PROGRAM PRG_TerminBoxInfo
VAR
END_VAR

//Terminal 0
GVL_IO.dwTerminalInfo[1].fbTerminalInfo(nTerminalState:= 8,
                                        sTerminalState => GVL_IO.dwTerminalInfo[0].sTerminalInfo);
//Terminal 1
GVL_IO.dwTerminalInfo[1].fbTerminalInfo(nTerminalState:= GVL_IO.dwTerminalInfo[1].nTerminal_State,
                                        sTerminalState => GVL_IO.dwTerminalInfo[1].sTerminalInfo);  
//Terminal 2
GVL_IO.dwTerminalInfo[2].fbTerminalInfo(nTerminalState:= GVL_IO.dwTerminalInfo[2].nTerminal_State,
                                        sTerminalState => GVL_IO.dwTerminalInfo[2].sTerminalInfo); 
//Terminal 3
GVL_IO.dwTerminalInfo[3].fbTerminalInfo(nTerminalState:= GVL_IO.dwTerminalInfo[3].nTerminal_State,
                                        sTerminalState => GVL_IO.dwTerminalInfo[3].sTerminalInfo); 
//Terminal 4
GVL_IO.dwTerminalInfo[4].fbTerminalInfo(nTerminalState:= GVL_IO.dwTerminalInfo[4].nTerminal_State,
                                        sTerminalState => GVL_IO.dwTerminalInfo[4].sTerminalInfo); 
//Terminal 5
GVL_IO.dwTerminalInfo[5].fbTerminalInfo(nTerminalState:= GVL_IO.dwTerminalInfo[5].nTerminal_State,
                                        sTerminalState => GVL_IO.dwTerminalInfo[5].sTerminalInfo); 
//Terminal 6
GVL_IO.dwTerminalInfo[6].fbTerminalInfo(nTerminalState:= GVL_IO.dwTerminalInfo[6].nTerminal_State,
                                        sTerminalState => GVL_IO.dwTerminalInfo[6].sTerminalInfo); 
//Terminal 7
GVL_IO.dwTerminalInfo[7].fbTerminalInfo(nTerminalState:= GVL_IO.dwTerminalInfo[7].nTerminal_State,
                                        sTerminalState => GVL_IO.dwTerminalInfo[7].sTerminalInfo); 
//Terminal 8
GVL_IO.dwTerminalInfo[8].fbTerminalInfo(nTerminalState:= GVL_IO.dwTerminalInfo[8].nTerminal_State,
                                        sTerminalState => GVL_IO.dwTerminalInfo[8].sTerminalInfo); 
//Terminal 9
GVL_IO.dwTerminalInfo[9].fbTerminalInfo(nTerminalState:= GVL_IO.dwTerminalInfo[9].nTerminal_State,
                                        sTerminalState => GVL_IO.dwTerminalInfo[9].sTerminalInfo); 
//Terminal 10
GVL_IO.dwTerminalInfo[10].fbTerminalInfo(nTerminalState:= GVL_IO.dwTerminalInfo[10].nTerminal_State,
                                        sTerminalState => GVL_IO.dwTerminalInfo[10].sTerminalInfo); 
//Terminal 11
GVL_IO.dwTerminalInfo[11].fbTerminalInfo(nTerminalState:= GVL_IO.dwTerminalInfo[11].nTerminal_State,
                                        sTerminalState => GVL_IO.dwTerminalInfo[11].sTerminalInfo); 
//Terminal 12
GVL_IO.dwTerminalInfo[12].fbTerminalInfo(nTerminalState:= GVL_IO.dwTerminalInfo[12].nTerminal_State,
                                        sTerminalState => GVL_IO.dwTerminalInfo[12].sTerminalInfo); 										
//Terminal 13
GVL_IO.dwTerminalInfo[13].fbTerminalInfo(nTerminalState:= GVL_IO.dwTerminalInfo[13].nTerminal_State,
                                        sTerminalState => GVL_IO.dwTerminalInfo[13].sTerminalInfo); 
//Terminal 14
GVL_IO.dwTerminalInfo[14].fbTerminalInfo(nTerminalState:= GVL_IO.dwTerminalInfo[14].nTerminal_State,
                                        sTerminalState => GVL_IO.dwTerminalInfo[14].sTerminalInfo);
										
//Terminal 15
GVL_IO.dwTerminalInfo[15].fbTerminalInfo(nTerminalState:= GVL_IO.dwTerminalInfo[15].nTerminal_State,
                                        sTerminalState => GVL_IO.dwTerminalInfo[15].sTerminalInfo); 
//Terminal 16
GVL_IO.dwTerminalInfo[16].fbTerminalInfo(nTerminalState:= 8,
                                        sTerminalState => GVL_IO.dwTerminalInfo[16].sTerminalInfo);										

//Terminal 17
GVL_IO.dwTerminalInfo[17].fbTerminalInfo(nTerminalState:= 8,
                                        sTerminalState => GVL_IO.dwTerminalInfo[17].sTerminalInfo);

//Terminal 18
GVL_IO.dwTerminalInfo[18].fbTerminalInfo(nTerminalState:= 8,
                                        sTerminalState => GVL_IO.dwTerminalInfo[18].sTerminalInfo);

//Terminal 19
GVL_IO.dwTerminalInfo[19].fbTerminalInfo(nTerminalState:= 8,
                                        sTerminalState => GVL_IO.dwTerminalInfo[19].sTerminalInfo);

//Terminal 20
GVL_IO.dwTerminalInfo[20].fbTerminalInfo(nTerminalState:= 8,
                                        sTerminalState => GVL_IO.dwTerminalInfo[20].sTerminalInfo);
																				
// Box 15
GVL_IO.dwBoxInfo[15].fbBoxInfo(nPnIoBoxState := GVL_IO.dwBoxInfo[15].nPnIoBoxState,    	
                               nPnIoBoxDiag  := GVL_IO.dwBoxInfo[15].nPnIoBoxDiag,
							   sBoxState      => GVL_IO.dwBoxInfo[15].sBoxState,
                               sBoxDiag       => GVL_IO.dwBoxInfo[15].sBoxDiag);
							   
//===========================================================================================================

END_PROGRAM

(* stored: Version 1.1.0.1, ProductVersion 3.1.4024.13
   POU PRG_TerminBoxInfo: Id {065a04fa-15dd-4ce4-b762-b796da589b85}, SpecialFunc None *)
